(* PLC project OOP_Curso, Beckhoff Automation GmbH TwinCAT PLC Control 3.5.13.21 *)
(* stored: creationDateTime 2023-05-27T11:18:57.8553898, modificationDateTime 2023-05-27T11:18:57.8622229 *)

INTERFACE I_Analog
METHOD Scale : BOOL
VAR_INPUT
END_VAR
END_METHOD
PROPERTY AnalogSignal : INT
END_PROPERTY
PROPERTY ScaledAnalog : INT
END_PROPERTY
END_INTERFACE

INTERFACE I_Run
METHOD Start : BOOL
VAR_INPUT
END_VAR
END_METHOD
METHOD Stop : BOOL
VAR_INPUT
END_VAR
END_METHOD
PROPERTY Coil : BOOL
END_PROPERTY
END_INTERFACE

PROGRAM _15_Interface_vs_Herencia
VAR
	//Nivel Sensor: 
	fbNivelSensor			: FB_NivelSensor;
	nNivelAnalogSensor 		: INT := 8000;
	nScaledNivelSensor 		: INT;
	nSensorNivelMaxValue 	: INT;

	//UltraSonidos
	fbUltraSonic 			: FB_UltraSonicSensor;
	nAnalogSensor 			: INT := 8000;
	nScaledSensor 			: INT;
	nSensorMaxValue 		: INT;
	
	//Variador de Frequencia
	fbVFD1 					: FB_VFD;
	bCoil1 					: BOOL;
	nFreqIn1  				: INT := 25;
	nFreqOut1 				: INT;	
	bStartVFD1 				: BOOL;
	
	//Pump
	fbPump1 				: FB_Pump;
	bCoilPump1				: BOOL;
	nFreqInPump1  			: INT := 25;
	nFreqOutPump1 			: INT;	
	bStartPump1 			: BOOL;	
END_VAR

            //Nivel Sensor
fbNivelSensor.AnalogSignal := nNivelAnalogSensor;
fbNivelSensor.MaxValue := 6;
nScaledNivelSensor := fbNivelSensor.ScaledAnalog;
fbNivelSensor.Scale();

//UltraSonidos
fbUltraSonic.AnalogSignal := nAnalogSensor;
fbUltraSonic.MaxValue := 6;
nScaledSensor := fbUltraSonic.ScaledAnalog;
fbUltraSonic.Scale();

//Variador de Frequencia
fbVFD1.AnalogSignal := nFreqIn1;
bCoil1 := fbVFD1.Coil;
nFreqOut1 := fbVFD1.ScaledAnalog;
fbVFD1.Scale();

IF bStartVFD1 THEN
	fbVFD1.Start();	
ELSE
	fbVFD1.Stop();
END_IF

//Pump
fbPump1.AnalogSignal := nFreqInPump1;
bCoilPump1 := fbPump1.Coil;
nFreqOutPump1 := fbPump1.ScaledAnalog;
fbPump1.Scale();

IF bStartPump1 THEN
	fbPump1.Start();	
ELSE
	fbPump1.Stop();
END_IF

          
END_PROGRAM

FUNCTION_BLOCK FB_NivelSensor IMPLEMENTS I_Analog
VAR_INPUT
END_VAR
VAR_OUTPUT
END_VAR
VAR
	_MaxValue 		: INT;
	_ScaledAnalog 	: INT;
	_AnalogSignal 	: INT;
END_VAR

            
          

{warning 'Agregar implementación de método'}
METHOD Scale : BOOL
                  ScaledAnalog := AnalogSignal * MaxValue / 1000;
                
END_METHOD

{warning 'Agregar implementación de propiedad'}
PROPERTY AnalogSignal : INT
GET
VAR
END_VAR
                    AnalogSignal := _AnalogSignal;
                  
END_GET
SET
VAR
END_VAR
                    _AnalogSignal := AnalogSignal;
                  
END_SET
END_PROPERTY

PROPERTY MaxValue : INT
GET
VAR
END_VAR
                    MaxValue := _MaxValue;
                  
END_GET
SET
VAR
END_VAR
                    _MaxValue := MaxValue;
                  
END_SET
END_PROPERTY

{warning 'Agregar implementación de propiedad'}
PROPERTY ScaledAnalog : INT
GET
VAR
END_VAR
                    ScaledAnalog := _ScaledAnalog;
                  
END_GET
SET
VAR
END_VAR
                    _ScaledAnalog := ScaledAnalog;
                  
END_SET
END_PROPERTY
END_FUNCTION_BLOCK

FUNCTION_BLOCK FB_Pump EXTENDS FB_VFD
VAR_INPUT
END_VAR
VAR_OUTPUT
END_VAR
VAR
END_VAR

            
          

{warning 'Agregar implementación de método'}
METHOD Scale : BOOL
                  ScaledAnalog := AnalogSignal * 100;
                
END_METHOD
END_FUNCTION_BLOCK

FUNCTION_BLOCK FB_UltraSonicSensor EXTENDS FB_NivelSensor
VAR_INPUT
END_VAR
VAR_OUTPUT
END_VAR
VAR

END_VAR

            
          

{warning 'Agregar implementación de método'}
METHOD Scale : BOOL
                  ScaledAnalog := AnalogSignal * MaxValue / 2000;
                
END_METHOD
END_FUNCTION_BLOCK

FUNCTION_BLOCK FB_VFD IMPLEMENTS I_Analog, I_Run
VAR_INPUT
END_VAR
VAR_OUTPUT
END_VAR
VAR
	_Coil 			: BOOL;
	_AnalogSignal 	: INT;
	_ScaledAnalog 	: INT;
END_VAR

            
          

{warning 'Agregar implementación de método'}
METHOD Scale : BOOL
                  ScaledAnalog := AnalogSignal * 200;
                
END_METHOD

{warning 'Agregar implementación de método'}
METHOD Start : BOOL
                  Coil := true;
                
END_METHOD

{warning 'Agregar implementación de método'}
METHOD Stop : BOOL
                  Coil := false;
                
END_METHOD

{warning 'Agregar implementación de propiedad'}
PROPERTY AnalogSignal : INT
GET
VAR
END_VAR
                    AnalogSignal := _AnalogSignal;
                  
END_GET
SET
VAR
END_VAR
                    _AnalogSignal := AnalogSignal;
                  
END_SET
END_PROPERTY

{warning 'Agregar implementación de propiedad'}
PROPERTY Coil : BOOL
GET
VAR
END_VAR
                    Coil := _Coil;
                  
END_GET
SET
VAR
END_VAR
                    _Coil := Coil;
                  
END_SET
END_PROPERTY

{warning 'Agregar implementación de propiedad'}
PROPERTY ScaledAnalog : INT
GET
VAR
END_VAR
                    ScaledAnalog := _ScaledAnalog;
                  
END_GET
SET
VAR
END_VAR
                    _ScaledAnalog := ScaledAnalog;
                  
END_SET
END_PROPERTY
END_FUNCTION_BLOCK
